PROGRAM Blinker
VAR
	TON2: TON;
	TON1: TON;
	t: BOOL;
	t2: BOOL;
END_VAR
VAR // added by the converter: edge detectors and wires of the graphical bodies
    _w1 : BOOL;
END_VAR

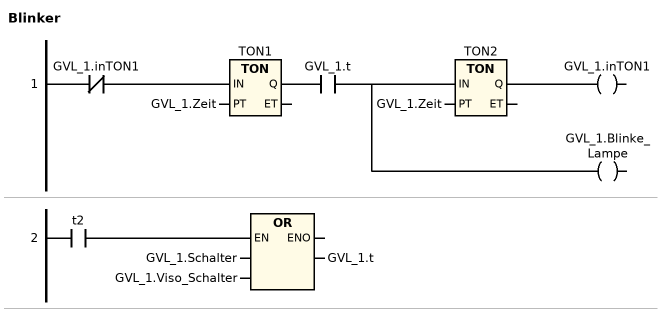
// NETWORK 1
TON1(IN := NOT GVL_1.inTON1, PT := GVL_1.Zeit); // TON
_w1 := TON1.Q AND GVL_1.t;
TON2(IN := _w1, PT := GVL_1.Zeit); // TON
GVL_1.inTON1 := TON2.Q;
GVL_1.Blinke_Lampe := _w1;

// NETWORK 2
IF t2 THEN GVL_1.t := GVL_1.Schalter OR GVL_1.Viso_Schalter; END_IF

END_PROGRAM

(* stored: Version 1.1.0.1, ProductVersion 3.1.4022.9
   POU Blinker: Id {6ed75c44-a9f5-441b-9b8e-dedff71b30a5}, SpecialFunc None *)
